FUNCTION_BLOCK Line (* openCV line drawer *)
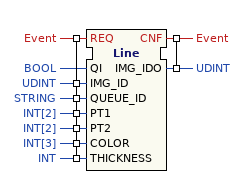
  EVENT_INPUT
    REQ WITH IMG_ID, QUEUE_ID, PT1, PT2, COLOR, THICKNESS;
  END_EVENT
  EVENT_OUTPUT
    CNF WITH IMG_IDO;
  END_EVENT
  VAR_INPUT
    QI : BOOL;
    IMG_ID : UDINT;
    QUEUE_ID : STRING;
    PT1 : ARRAY [0..1] OF INT;
    PT2 : ARRAY [0..1] OF INT;
    COLOR : ARRAY [0..2] OF INT;
    THICKNESS : INT;
  END_VAR
  VAR_OUTPUT
    IMG_IDO : UDINT;
  END_VAR
END_FUNCTION_BLOCK
